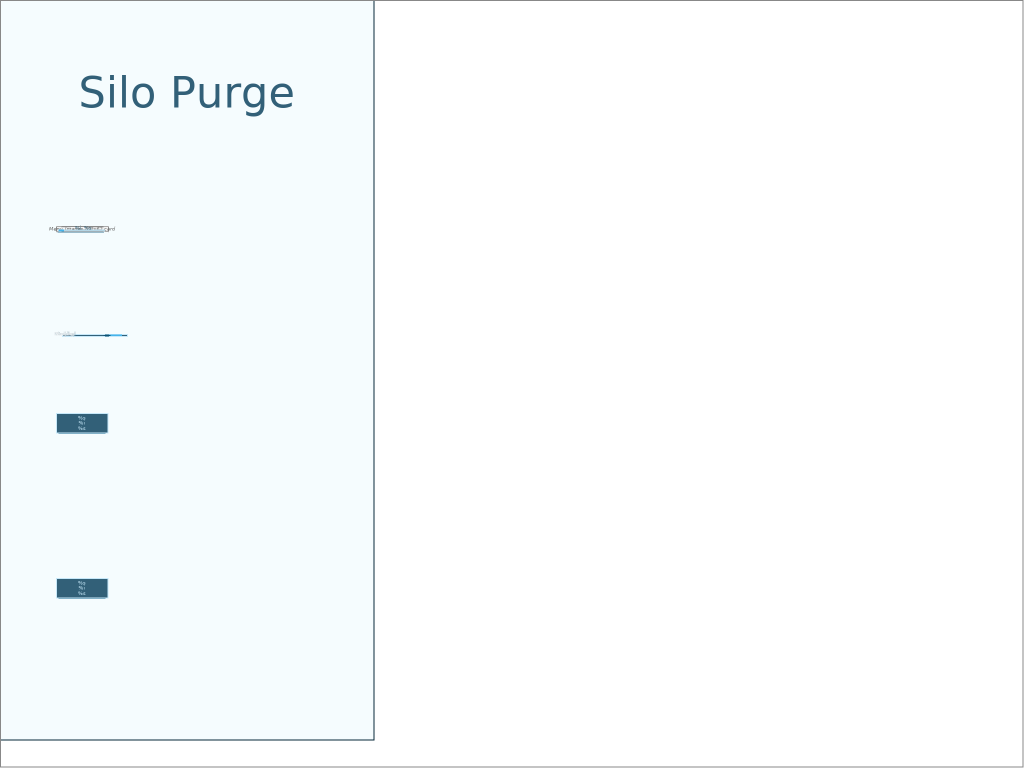
VISUALIZATION Purge  // 1024x768
VAR_INPUT
	xSELECTED: BOOL;
	Hover_X: UINT;
END_VAR
VAR
	Hover_Y: UINT;
END_VAR
    Rectangle (0,0 374x740)
    Frame (62,334 255x45)
        shows f_Checkbox(Setting := prvars.purge_enabled, fb_ref := Test_PRG.test_toggle, Name := 'Enabled', Hover := Hover_X = 0 AND Hover_Y = 0, Selected := Hover_X = 0 AND Hover_Y = 0 AND xSelected)
    Frame (56,413 267x130)
        shows Setting_Card_Frame(Setting := prvars.purge_frequency, Hover := Hover_X = 0 AND Hover_Y = 1, Selected := Hover_X = 0 AND Hover_Y = 1 AND xSelected, ui_Increment := 100, Max_Value := 10000, Min_Value := 100, Name := 'purge every', Units := 'gallons pumped')
    Frame (56,578 267x130)
        shows Setting_Card_Frame(Setting := prvars.purge_duration, Hover := Hover_X = 0 AND Hover_Y = 2, Selected := Hover_X = 0 AND Hover_Y = 2 AND xSelected, ui_Increment := 1, Max_Value := 100, Min_Value := 1, Name := 'purge for', Units := 'seconds')
    Frame (56,226 267x74)
        shows f_ProgressBar(Value := Test_PRG.Purge_Control.Cycle_Volume, Percentage := TO_UINT(TO_REAL((Test_PRG.Purge_Control.Cycle_Volume) / TO_REAL(Test_PRG.Purge_Control.Gallons_Setpoint)) * 100), Units := 'gal.')
    Rectangle (0,0 374x185), "Silo Purge"
    hotkey  Id=481041580032, Key=KeyDown=True, KeyName=left, ActionToExecute=Action=STSnippet=IF xSelected THEN RETURN; END_IF IF Hover_X = 0 THEN IF Hover_Y < 2 THEN Hover_Y:= Hover_Y + 1; END_IF END_IF IF Hover_X = 1 THEN IF Hover_Y < 5 THEN Hover_Y:= Hover_Y + 1; END_IF END_IF, VisuElemId=-1
    hotkey  Id=481040531456, Key=KeyDown=True, KeyName=right, ActionToExecute=Action=STSnippet=IF xSelected THEN RETURN; END_IF IF Hover_Y > 0 THEN Hover_Y:= Hover_Y - 1; END_IF, VisuElemId=-1
END_VISUALIZATION

// CR1104/Application/HMI/Components/Pages/Settings
VISUALIZATION Settings  // 1024x768
END_VISUALIZATION

// CR1104/Application/HMI/Components/Setting Card/Test_Card
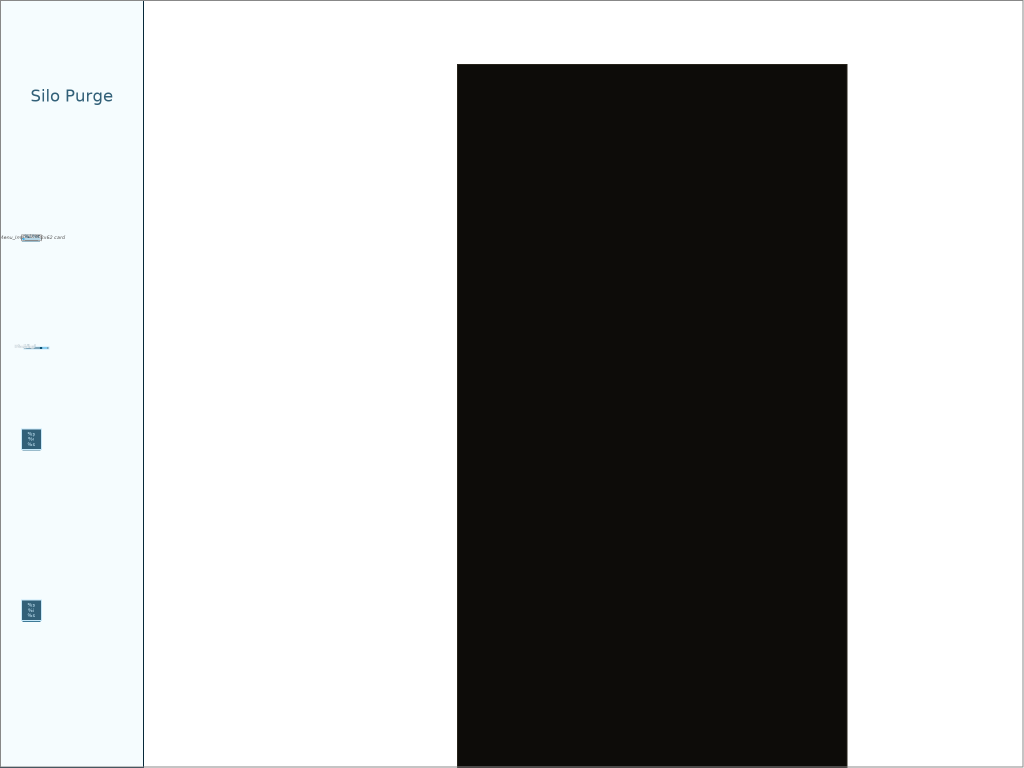
VISUALIZATION Test_Card  // 1024x768
VAR
	Navigate: Keypad_Navigation_FB:= (
					X_items:= 2, 
					Y_Items:= 1
				);
END_VAR
    RoundedRectangle (457,64 390x794), colour toggle: Navigate.Position_X = 0
        p3560616238: TO_INT(Navigate.Position_X = 1) * (-126)
    Frame (0,0 393x797)
        shows Purge()
    hotkey  Id=481037385728, Key=KeyDown=True, KeyName=right, ActionToExecute=Action=STSnippet=Navigate.up();, VisuElemId=-1
    hotkey  Id=481038434304, Key=KeyDown=True, KeyName=left, ActionToExecute=Action=STSnippet=Navigate.down();, VisuElemId=-1
    hotkey  Id=481039482880, Key=KeyDown=True, KeyName=up, ActionToExecute=Action=STSnippet=Navigate.left();, VisuElemId=-1
    hotkey  Id=481040531456, Key=KeyDown=True, KeyName=down, ActionToExecute=Action=STSnippet=Navigate.right();, VisuElemId=-1
END_VISUALIZATION

// CR1104/Application/HMI/Components/POUs/Hotkey/Tank_Frame
VISUALIZATION Tank_Frame  // 1024x768
END_VISUALIZATION

// CR1104/Application/HMI/Components/Setting Card/Visus/Setting_Card_Frame
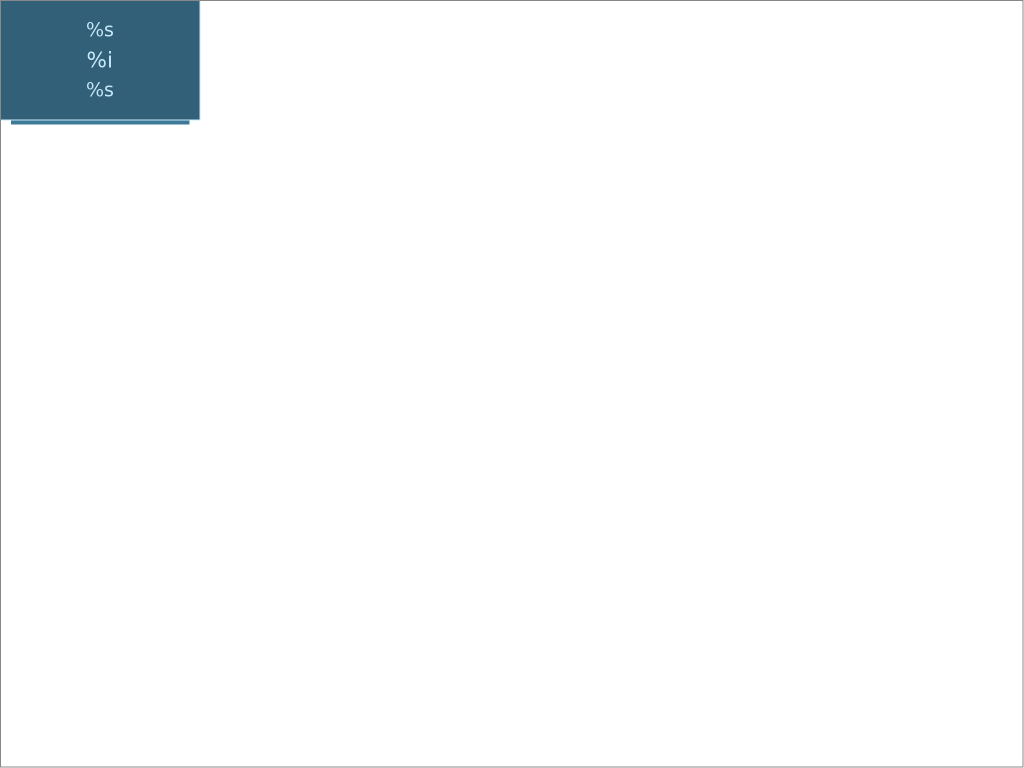
VISUALIZATION Setting_Card_Frame  // 1024x768
///
VAR_IN_OUT
	Setting: UINT;
END_VAR
///
VAR_INPUT
	Hover: BOOL;
	Selected: BOOL;
	ui_Increment: UINT:= 1;
	Max_Value: UINT;
	Min_Value: UINT;
	Name: STRING;
	Units: STRING;
END_VAR
///
VAR
	Setting_Card: fb_Setting_Card;
END_VAR
///
    RoundedRectangle (11,67 178x57)
    Rectangle (0,0 200x120)
    Rectangle (0,0 200x120), invisible if: NOT(Hover)
    Rectangle (1,15 200x30), "%s", text variable: Name
    Rectangle (1,75 200x30), "%s", text variable: Units
    Rectangle (1,45 200x30), "%i", text variable: Setting
    Rectangle (0,0 200x120), invisible if: NOT(Selected)
    Rectangle (0,75 200x30), "%s", text variable: Units, invisible if: NOT(Selected)
    Rectangle (0,15 200x30), "%s", text variable: Name, invisible if: NOT(Selected)
    Rectangle (0,45 200x30), "%i", text variable: Setting, invisible if: NOT(Selected)
    hotkey  Id=481037385728, Key=KeyDown=True, KeyName=right, ActionToExecute=Action=STSnippet=IF NOT Selected THEN RETURN; END_IF Setting_Card(Value:= Setting, increment:= ui_increment, maximum:= Max_Value, minimum:= Min_Value,); Setting_Card.increase(); //Setting_Card(Value:= Setting);, VisuElemId=-1
    hotkey  Id=481038434304, Key=KeyDown=True, KeyName=left, ActionToExecute=Action=STSnippet=IF NOT Selected THEN RETURN; END_IF Setting_Card(Value:= Setting, increment:= ui_increment, maximum:= Max_Value, minimum:= Min_Value,); Setting_Card.decrease(); //Setting_Card(Value:= Setting);, VisuElemId=-1
END_VISUALIZATION
